Yaskawa INFORM job: R1_W73(0,-90)KM-OK.JBI

/JOB
//NAME R1_W73(0,-90)KM-OK
///FOLDERNAME KRIS-SCIANA
//POS
///NPOS 128,128,0,5,0,0
///TOOL 0
///POSTYPE PULSE
///PULSE
C00000=-40404,-32975,-87125,-16022,87663,5338
C00001=-149842,-73226,-111008,-16022,94395,5338
C00002=-196430,-28535,-98412,17908,105328,15740
C00003=-197819,-28541,-95016,18260,103548,15106
C00004=-200339,-28643,-93145,19132,102819,14321
C00005=-200339,-29850,-92907,19066,102093,14204
C00006=-198353,-28437,-93612,18398,102863,14858
C00007=-194160,-43345,-101472,6781,97426,15909
C00008=-194408,-42587,-101034,6883,97560,15852
C00009=-193796,-43946,-102216,6636,97553,16011
C00010=-201919,-14623,-81254,29586,105679,13958
C00011=-201296,-13906,-80720,29363,105554,14109
C00012=-202898,-15552,-82103,29953,105971,13746
C00013=-202564,-15340,-83288,29973,106616,14022
C00014=-201706,-14587,-86146,30041,108271,14729
C00015=-194060,1523,-76765,18551,116913,19891
C00016=-194060,-226,-76587,18372,115954,19725
C00017=-196031,-5339,-80231,20914,112748,19532
C00018=-197990,-8736,-83028,21568,113067,19065
C00019=-197425,-9792,-82211,21200,111990,19009
C00020=-196969,-9135,-81776,21059,111976,19132
C00021=-197863,-8882,-82791,21487,112841,19056
C00022=-189091,-8045,-83877,18664,112431,21315
C00023=-189216,-11043,-83213,18430,110597,20976
C00024=-189216,-12280,-83029,18331,109883,20859
C00025=-189216,-11043,-83213,18430,110597,20976
C00026=-187860,-13057,-85333,17999,110646,21345
C00027=-187738,-15527,-85495,17806,109510,21198
C00028=-188240,-14336,-84615,17987,109655,21087
C00029=-187877,-14602,-87082,18044,110918,21384
C00030=-202564,-15340,-83288,29973,106616,14022
C00031=-180747,-34566,-103569,5865,76463,-74344
C00032=-3241,-154154,-132855,1912,-2104,-59891
C00033=90131,-154154,-132855,1912,25799,-59891
C00034=133217,-9267,-70818,-4736,81507,-40311
C00035=147446,66185,-7865,-6124,89018,-32930
C00036=146775,67981,670,-5813,84671,-32906
C00037=142065,101170,34317,5326,97892,-38868
C00038=142065,100549,34406,5321,97520,-38885
C00039=142065,101170,34317,5326,97892,-38868
C00040=146775,67981,670,-5813,84671,-32906
C00041=141709,70703,3575,5716,88259,-35170
C00042=142000,70934,3857,5588,88189,-35093
C00043=141709,70505,3632,5716,88123,-35177
C00044=141466,75678,7759,5822,88256,-35240
C00045=150714,57521,-9985,-12467,84539,-31420
C00046=152456,58301,-6639,-13350,83146,-30782
C00047=152350,58936,-5903,-13300,83008,-30798
C00048=152043,57091,-7724,-13148,83136,-30899
C00049=150714,57521,-9985,-12467,84539,-31420
C00050=150397,65709,-1678,-12325,83616,-31417
C00051=152081,83448,18494,-17729,87965,-36105
C00052=145309,67853,4255,2462,78780,-48595
C00053=142342,76526,12204,14792,84634,-59311
C00054=139855,76006,10433,20657,83547,-58718
C00055=138944,70547,-13352,-2713,109632,-82660
C00056=150992,69723,-1355,-37332,105967,-89594
C00057=150476,128390,79342,-39456,121713,-63684
C00058=149946,126808,77134,-37730,123094,-66135
C00059=150687,93176,30567,-40025,118220,-86305
C00060=151970,82147,17677,-42167,111883,-84378
C00061=150687,93185,30564,-40027,118225,-86307
C00062=152182,83304,17941,-42342,112294,-84475
C00063=151694,72284,4221,-38531,106791,-89962
C00064=151393,70428,3257,-38368,106391,-89923
C00065=150986,73664,7109,-38113,105680,-89808
C00066=151161,78896,6636,-38820,108108,-90659
C00067=150730,108324,43859,-37200,101741,-88479
C00068=138109,93543,17707,-11473,100978,-85696
C00069=126155,75677,-665,13089,94512,-81960
C00070=136360,44466,-35259,-6214,94815,-84020
C00071=129275,89679,9974,19452,120712,-90755
C00072=124685,94998,28008,29047,119888,-86461
C00073=125807,95110,28281,28956,119459,-86150
C00074=125255,100992,28971,31279,121490,-85312
C00075=130721,42993,-42514,6818,104896,-53830
C00076=133217,-9267,-70818,-4736,81507,-40311
C00077=90131,-154154,-132855,1912,25799,-59891
C00078=-27662,-161693,-134781,-6409,23242,-55851
C00079=-153837,-124252,-132652,-6394,34053,-55850
C00080=-180749,-57313,-97512,6480,61132,-75141
C00081=-181681,-58157,-94543,7323,58956,-75591
C00082=-180203,-60166,-93803,6313,57366,-75174
C00083=-181915,-57690,-94240,7494,59028,-75667
C00084=-183086,-60514,-94424,8485,57804,-76167
C00085=-183688,-52020,-90180,8774,59600,-76232
C00086=-183472,-54404,-92153,8618,59567,-76163
C00087=-194372,-19965,-77328,28851,83810,-77840
C00088=-194352,-19726,-77485,28832,83998,-77787
C00089=-192839,-24502,-80432,28081,83025,-77568
C00090=-192267,-26347,-80544,27830,82091,-77618
C00091=-192787,-23975,-80802,28033,83453,-77448
C00092=-193865,-26434,-81106,28635,82790,-77939
C00093=-190854,-30389,-83029,27131,81227,-77386
C00094=-191509,-27758,-83155,27393,82677,-77248
C00095=-191676,-23479,-84120,27380,85212,-76702
C00096=-161879,-68419,-121263,-50083,88779,-73415
C00097=-161876,-91492,-113119,-51274,77787,-67446
C00098=-164907,-89219,-108956,-50337,75324,-67571
C00099=-164989,-85960,-105925,-50342,75158,-67521
C00100=-166079,-87440,-108199,-49792,75019,-67981
C00101=-164680,-90458,-107994,-50658,74641,-67078
C00102=-166572,-90913,-107959,-49982,73492,-67393
C00103=-165515,-88688,-108094,-50145,74844,-67608
C00104=-167050,-87345,-105736,-37517,58682,-66535
C00105=-167580,-87197,-104728,-37395,58030,-66518
C00106=-167739,-85864,-105828,-36810,59062,-66997
C00107=-166381,-88790,-105608,-38219,58303,-66072
C00108=-167025,-85240,-103855,-37559,58631,-66501
C00109=-166590,-87652,-106603,-37658,59170,-66520
C00110=-163660,-90098,-110841,-38913,61454,-66120
C00111=-163662,-68991,-119593,-35124,74591,-70861
C00112=-164323,-67552,-119186,-34656,74786,-71140
C00113=-42611,-72193,-121247,-35066,73992,-70748
C00114=-42611,-136501,-121247,37840,71925,-70748
C00115=30194,-138584,-136989,36596,19750,-68315
C00116=30194,-138584,-136989,36596,19750,-68315
C00117=48317,-32494,-96788,-15754,91861,-54663
C00118=38193,-30329,-90168,-1738,86717,-61333
C00119=37412,-28378,-87220,-1336,85895,-61525
C00120=40911,-29532,-88262,-3131,86017,-60613
C00121=58834,66382,-3921,-1467,93638,-45665
C00122=61274,64840,-6146,-2451,94263,-45016
C00123=60162,91684,24560,8859,97426,-41962
C00124=59447,93093,21113,9166,100305,-41958
C00125=54612,98200,13834,4767,109112,-43277
C00126=53873,97111,13222,4370,109077,-43421
C00127=-37947,-148118,-122898,-84151,100970,-75634
BC00000=86652,945,1075157
BC00001=383249,913,1075157
BC00002=398174,90672,1075175
BC00003=398174,94386,1075175
BC00004=398174,95871,1075175
BC00005=398174,95871,1075175
BC00006=398174,95871,1075175
BC00007=398174,107607,1075175
BC00008=398174,107607,1075175
BC00009=398174,107607,1075175
BC00010=398174,86976,1075175
BC00011=398174,86976,1075175
BC00012=398174,86976,1075175
BC00013=398174,85141,1075175
BC00014=398174,80554,1075175
BC00015=398174,80554,1075175
BC00016=398174,80554,1075175
BC00017=398174,80554,1075175
BC00018=398174,80554,1075175
BC00019=398174,80554,1075175
BC00020=398174,80554,1075175
BC00021=398174,80554,1075175
BC00022=398174,80554,1075175
BC00023=398174,80554,1075175
BC00024=398174,80554,1075175
BC00025=398174,80554,1075175
BC00026=398174,80554,1075175
BC00027=398174,80554,1075175
BC00028=398174,80554,1075175
BC00029=398174,80554,1075175
BC00030=398174,85141,1075175
BC00031=398174,58980,1075175
BC00032=129287,13301,1075175
BC00033=129287,433299,1075175
BC00034=251623,516237,1075175
BC00035=299173,515631,1075175
BC00036=299173,515631,1075175
BC00037=299173,515631,1075175
BC00038=299173,515631,1075175
BC00039=299173,515631,1075175
BC00040=299173,515631,1075175
BC00041=299173,515631,1075175
BC00042=299173,515631,1075175
BC00043=299173,515631,1075175
BC00044=299173,515631,1075175
BC00045=299173,515631,1075175
BC00046=299173,515631,1075175
BC00047=299173,515631,1075175
BC00048=299173,515631,1075175
BC00049=299173,515631,1075175
BC00050=299173,515631,1075175
BC00051=299173,515631,1075175
BC00052=299173,515631,1075175
BC00053=299173,515632,1075173
BC00054=299173,515631,1075175
BC00055=236130,485794,1075175
BC00056=236130,485794,1075175
BC00057=236130,478839,1075175
BC00058=236130,478839,1075175
BC00059=236130,478839,1075175
BC00060=236130,478839,1075175
BC00061=236130,478839,1075175
BC00062=236130,478839,1075175
BC00063=236130,478839,1075175
BC00064=236130,478839,1075175
BC00065=236130,478839,1075175
BC00066=236130,478839,1075175
BC00067=236130,478839,1075175
BC00068=236130,478839,1075175
BC00069=236130,478839,1075175
BC00070=236130,478839,1075175
BC00071=236130,478839,1075175
BC00072=236130,478839,1075175
BC00073=236130,478839,1075175
BC00074=236130,478839,1075175
BC00075=246766,504514,1075175
BC00076=251623,516237,1075175
BC00077=129287,433299,1075175
BC00078=132935,44385,1075175
BC00079=397875,59424,1075173
BC00080=398174,58966,1075175
BC00081=398174,63329,1075175
BC00082=398174,65074,1075175
BC00083=398174,65074,1075175
BC00084=398174,65074,1075175
BC00085=398174,65113,1075175
BC00086=398174,64241,1075175
BC00087=398174,59338,1075175
BC00088=398174,58794,1075175
BC00089=398174,58749,1075175
BC00090=398174,59838,1075175
BC00091=398174,59838,1075175
BC00092=398174,59838,1075175
BC00093=398174,59797,1075175
BC00094=398174,58061,1075175
BC00095=398174,53722,1075175
BC00096=398174,135435,1075175
BC00097=398174,135422,1075175
BC00098=398174,134136,1075175
BC00099=398174,133622,1075175
BC00100=398174,133622,1075175
BC00101=398174,133622,1075175
BC00102=398174,133622,1075175
BC00103=398174,130807,1075175
BC00104=398174,103027,1075175
BC00105=398174,103038,1075175
BC00106=398174,103038,1075175
BC00107=398174,103038,1075175
BC00108=398174,106110,1075175
BC00109=398174,105557,1075175
BC00110=398174,104176,1075175
BC00111=398174,104190,1075175
BC00112=176805,33,1075175
BC00113=68317,33,1075175
BC00114=68317,33,1075175
BC00115=68317,33,1075175
BC00116=70991,324077,1075175
BC00117=70991,324077,1075175
BC00118=70991,324077,1075175
BC00119=70991,324077,1075175
BC00120=70991,324077,1075175
BC00121=36742,425083,1075175
BC00122=36742,425083,1075175
BC00123=36742,444685,1075175
BC00124=36742,444685,1075175
BC00125=46495,445330,1075175
BC00126=48059,443707,1075175
BC00127=233905,457726,1075173
///POSTYPE BASE
///RECTAN
///RCONF 0,0,0,0,1,0,0,0,0,0,0,0,0,0,0,0,0,0,0,0,0,0,0,0
P00006=2.006,1.622,-0.565,0.0000,0.0000,0.0000
///RCONF 0,0,0,0,0,0,0,0,0,0,0,0,0,0,0,0,0,0,0,0,0,0,0,0
P00023=-2.957,-4.083,2.762,0.0000,0.0000,0.0000
P00024=-1.466,-0.226,-0.419,0.0000,0.0000,0.0000
P00025=3.643,0.007,-2.585,0.0000,0.0000,0.0000
P00026=2.644,0.055,-2.583,0.0000,0.0000,0.0000
//INST
///DATE 2025/04/02 09:13
///ATTR SC,RW
///GROUP1 RB1,BS1
NOP
'r1_W73(0,-90)
SFTOF
MOVL C00000 BC00000 V=833.3
MOVL C00001 BC00001 V=833.3
MOVL C00002 BC00002 V=500.0
MOVL C00003 BC00003 V=250.0
MOVL C00004 BC00004 V=133.3
REFP 3 C00005 BC00005
CALL JOB:SEARCH-R1
SET P023 P006
SFTON P023
MOVL C00006 BC00006 V=60.0
MOVL C00007 BC00007 V=60.0
REFP 3 C00008 BC00008
CALL JOB:SEARCH-R1
SET P023 P006
SFTON P023
MOVL C00009 BC00009 V=60.0
MOVL C00010 BC00010 V=60.0
REFP 3 C00011 BC00011
CALL JOB:SEARCH-R1
SET P023 P006
SFTON P023
MOVL C00012 BC00012 V=60.0
MOVL C00013 BC00013 V=166.7
MOVL C00014 BC00014 V=166.7
'Path W514
SFTOF
MOVL C00015 BC00015 V=60.0
REFP 3 C00016 BC00016
CALL JOB:SEARCH-R1
SET P025 P006
SFTON P025
MOVL C00017 BC00017 V=60.0
MOVL C00018 BC00018 V=60.0
MOVL C00019 BC00019 V=60.0
REFP 3 C00020 BC00020
CALL JOB:SEARCH-R1
SET P025 P006
SFTOF
MOVL C00021 BC00021 V=60.0
MOVL C00022 BC00022 V=166.7
MOVL C00023 BC00023 V=60.0
REFP 3 C00024 BC00024
CALL JOB:SEARCH-R1
SET P026 P006
SFTON P026
MOVL C00025 BC00025 V=60.0
MOVL C00026 BC00026 V=60.0
MOVL C00027 BC00027 V=60.0
REFP 3 C00028 BC00028
CALL JOB:SEARCH-R1
SET P026 P006
SFTOF
MOVL C00029 BC00029 V=60.0
MOVL C00030 BC00030 V=166.7
SFTON P023
MOVJ C00031 BC00031 VJ=100.00
'POMIAR 2 STRONA
'Path S1141
SFTOF
MOVJ C00032 BC00032 VJ=100.00
MOVJ C00033 BC00033 VJ=100.00
MOVJ C00034 BC00034 VJ=100.00
MOVJ C00035 BC00035 VJ=100.00
MOVL C00036 BC00036 V=100.0
MOVL C00037 BC00037 V=60.0
REFP 3 C00038 BC00038
CALL JOB:SEARCH-R1
SET P024 P006
SFTON P024
MOVL C00039 BC00039 V=60.0
MOVL C00040 BC00040 V=100.0
MOVL C00041 BC00041 V=60.0
REFP 3 C00042 BC00042
CALL JOB:SEARCH-R1
SET P024 P006
SFTON P024
MOVL C00043 BC00043 V=60.0
MOVL C00044 BC00044 V=100.0
MOVL C00045 BC00045 V=100.0
MOVL C00046 BC00046 V=60.0
REFP 3 C00047 BC00047
CALL JOB:SEARCH-R1
SET P024 P006
SFTON P024
MOVL C00048 BC00048 V=60.0
MOVL C00049 BC00049 V=100.0
MOVL C00050 BC00050 V=100.0
CALL JOB:COFNIJ_DRUT
SFTOF
SFTOF
SFTON P024
MOVL C00051 BC00051 V=100.0 PL=0
MACRO1 MJ#(0) ARGF12
ARCON
MOVL C00052 BC00052 V=9.2
MOVL C00053 BC00053 V=9.2
ARCOF
MOVL C00054 BC00054 V=100.0
MOVL C00055 BC00055 V=100.0
MOVJ C00056 BC00056 VJ=100.00
'COMMENT
'COMMENT
SFTOF
SFTON P024
MOVL C00057 BC00057 V=100.0
MOVL C00058 BC00058 V=100.0 PL=0
MACRO1 MJ#(0) ARGF12
ARCON
MOVL C00059 BC00059 V=8.3
ARCOF
MOVL C00060 BC00060 V=33.3
ARCON
MOVL C00061 BC00061 V=9.2
ARCOF
MOVL C00062 BC00062 V=100.0
MOVL C00063 BC00063 V=100.0
'COMMENT
'COMMENT
SFTOF
SFTON P024
MOVL C00064 BC00064 V=100.0 PL=0
MACRO1 MJ#(0) ARGF12
ARCON
MOVL C00065 BC00065 V=9.2
ARCOF
MOVL C00066 BC00066 V=100.0
MOVJ C00067 BC00067 VJ=100.00
MOVJ C00068 BC00068 VJ=100.00
MOVJ C00069 BC00069 VJ=100.00
MOVJ C00070 BC00070 VJ=100.00
MOVJ C00071 BC00071 VJ=100.00
'COMMENT
'COMMENT
SFTOF
SFTON P024
MOVL C00072 BC00072 V=100.0 PL=0
MACRO1 MJ#(0) ARGF12
ARCON
MOVL C00073 BC00073 V=11.7
ARCOF
MOVL C00074 BC00074 V=100.0
SFTOF
MOVJ C00075 BC00075 VJ=100.00
MOVJ C00076 BC00076 VJ=100.00
MOVJ C00077 BC00077 VJ=100.00
MOVJ C00078 BC00078 VJ=100.00
MOVJ C00079 BC00079 VJ=100.00
'KONIEC POMIAR 2 STRONA
MOVL C00080 BC00080 V=166.7
MOVL C00081 BC00081 V=166.7
SFTON P023
MOVL C00082 BC00082 V=100.0 PL=0
REFP 1 C00083 BC00083
REFP 2 C00084 BC00084
MACRO1 MJ#(0) ARGF12
ARCON
MOVL C00085 BC00085 V=9.2
ARCOF
MOVL C00086 BC00086 V=100.0
SFTOF
MOVL C00087 BC00087 V=100.0
MOVL C00088 BC00088 V=100.0
SFTON P026
MOVL C00089 BC00089 V=100.0
MOVL C00090 BC00090 V=100.0 PL=0
REFP 1 C00091 BC00091
REFP 2 C00092 BC00092
MACRO1 MJ#(0) ARGF12
ARCON
MOVL C00093 BC00093 V=9.2
ARCOF
MOVL C00094 BC00094 V=166.7
MOVL C00095 BC00095 V=166.7
SFTOF
'Path W513
SFTOF
SFTON P023
MOVJ C00096 BC00096 VJ=100.00
MOVL C00097 BC00097 V=166.7
MOVL C00098 BC00098 V=166.7
MOVL C00099 BC00099 V=100.0 PL=0
REFP 1 C00100 BC00100
REFP 2 C00101 BC00101
MACRO1 MJ#(0) ARGF12
ARCON
MOVL C00102 BC00102 V=9.5
ARCOF
MOVL C00103 BC00103 V=100.0
MOVL C00104 BC00104 V=100.0
MOVL C00105 BC00105 V=100.0 PL=0
REFP 1 C00106 BC00106
REFP 2 C00107 BC00107
MACRO1 MJ#(0) ARGF12
ARCON
MOVL C00108 BC00108 V=9.5
ARCOF
MOVL C00109 BC00109 V=166.7
MOVL C00110 BC00110 V=166.7
MOVL C00111 BC00111 V=166.7
SFTOF
MOVJ C00112 BC00112 VJ=50.00
MOVJ C00113 BC00113 VJ=50.00
MOVJ C00114 BC00114 VJ=50.00
MOVJ C00115 BC00115 VJ=50.00
MOVJ C00116 BC00116 VJ=50.00
SFTOF
MOVJ C00117 BC00117 VJ=100.00
SFTON P026
MACRO1 MJ#(0) ARGF12
MOVJ C00118 BC00118 VJ=50.00
MOVL C00119 BC00119 V=166.7 PL=0
ARCON
MOVL C00120 BC00120 V=9.2
MOVL C00121 BC00121 V=9.2
SFTON P025
MOVL C00122 BC00122 V=9.2
MOVL C00123 BC00123 V=9.2
ARCOF
MOVJ C00124 BC00124 VJ=100.00
SFTOF
MOVJ C00125 BC00125 VJ=100.00
MOVJ C00126 BC00126 VJ=100.00
MOVJ C00127 BC00127 VJ=100.00
END
